// TIA Portal V21 export
// export: Created 2026-07-07T09:15:55.8352405Z, ExportSetting WithReadOnly, DisplayName Totally Integrated Automation Portal, DisplayVersion V21, DisplayName SINAMICS Startdrive Advanced, DisplayVersion V21, DisplayName SINAMICS Startdrive G110M, G120, G120C, G120D, G120P, G115D, DisplayVersion V21, DisplayName SINAMICS Startdrive G130, G150, S120, S150, G200, G220, S200, S210, S220, Innomotics MVD, DisplayVersion V21, DisplayName STEP 7 Professional, DisplayVersion V21, DisplayName STEP 7 Safety, DisplayVersion V21, DisplayName Tech WebApplication, DisplayVersion V21, DisplayName WinCC Basic/Comfort/Advanced, DisplayVersion V21, DisplayName WinCC Professional, DisplayVersion V21, DisplayName WinCC Unified, DisplayVersion V21
Screen "Screen_01_MainOverview"  Nonex480, Template=模板_1
  ScreenLayer 
    TextField "Title" at 20,12 size 760x34  Text="画面 1：主监控画面"
    TextField "NavBar" at 20,430 size 760x34  Text="主监控 手动调试 参数设置 报警诊断 趋势"
    TextField "Hdr_EC_pH_288" at 20,60 size 360x26  Text="EC / pH 总览"
    TextField "Body_EC_pH_304" at 20,84 size 360x126  Text="EC_Set_SP | EC_Actual | pH_Set_SP | pH_Actual | Active_EC_SP | Active_pH_SP | Growth_Stage"
    TextField "Hdr_Item_320" at 410,60 size 370x26  Text="系统状态"
    TextField "Body_Item_336" at 410,84 size 370x126  Text="Remote_Comms_OK | Comm_Normal | System_Alarm_Light | Emergency_Stop | Manual_Active | Auto_Active"
    TextField "Hdr_Item_352" at 20,225 size 360x26  Text="执行量监控"
    TextField "Body_Item_368" at 20,249 size 360x126  Text="q_f_cmd | q_a_cmd | Valve_F_Actual | Valve_A_Actual | AQ_Valve_F_Raw | AQ_Valve_A_Raw"
    TextField "Hdr_Item_384" at 410,225 size 370x26  Text="多通道输出"
    TextField "Body_Item_400" at 410,249 size 370x126  Text="q_n_cmd | q_p_cmd | q_k_cmd | Stage_EC_SP | Stage_pH_SP | Setpoint_Protection_Active"
